{attribute 'qualified_only'}
VAR_GLOBAL CONSTANT
    nGRID_SCAN_POINT_WINDOW_MIN : INT := 0;
    nGRID_SCAN_POINT_WINDOW_MAX : INT := 10;
END_VAR

(* stored: Version 1.1.0.1
   GVL Constants: Id {68d21a5d-b6f1-458e-a6b3-1dca277ea9c6} *)
